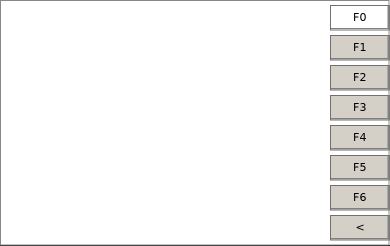
VISUALIZATION VPP  // 390x246
    Button (330,5 60x25), "F0"
    Button (330,35 60x25), "F1"
    Button (330,65 60x25), "F2"
    Button (330,95 60x25), "F3"
    Button (330,125 60x25), "F4"
    Button (330,155 60x25), "F5"
    Button (330,185 60x25), "F6"
    Line (0,245) (390,245)
    Button (330,215 60x25), "<"
        OnMouseClick: change screen: V_Safety
END_VISUALIZATION

(* stored: Version 1.1.0.1, ProductVersion 3.1.4024.9
   Visu VPP: Id {98cd63f7-24ec-4f71-a506-baa623a97061} *)
